INTERFACE I_XTS_Mover_PLC EXTENDS I_CH_Object

{attribute 'OPC.UA.DA.Property' := '1'}
{attribute 'monitoring':='call'}
PROPERTY DefaultAcceleration : LREAL
GET
END_GET
SET
END_SET
END_PROPERTY

{attribute 'OPC.UA.DA.Property' := '1'}
{attribute 'monitoring':='call'}
PROPERTY DefaultDeceleration : LREAL
GET
END_GET
SET
END_SET
END_PROPERTY

{attribute 'OPC.UA.DA.Property' := '1'}
{attribute 'monitoring':='call'}
PROPERTY DefaultJerk : LREAL
GET
END_GET
SET
END_SET
END_PROPERTY

{attribute 'monitoring':='call'}
PROPERTY DrivenDistance : LREAL
GET
END_GET
END_PROPERTY

(*The _ PLC interface provides the user with a simplified interface for commanding between the stations. Sometimes, however, this is not enough. 
Either you get the corresponding interface with the __Queryinterface or you can get full access with this property.*)
PROPERTY FullAccess : I_XTS_Mover
GET
END_GET
END_PROPERTY

{attribute 'monitoring':='call'}
PROPERTY LagDistance : LREAL
GET
END_GET
END_PROPERTY

{attribute 'monitoring':='call'}
PROPERTY LastCmdTargedGap : LREAL
GET
END_GET
END_PROPERTY

{attribute 'monitoring':='call'}
PROPERTY LUID : STRING
GET
END_GET
END_PROPERTY

{attribute 'monitoring':='call'}
PROPERTY PositionOnTrack : LREAL
GET
END_GET
END_PROPERTY

{attribute 'monitoring':='call'}
PROPERTY PUBLIC ProductData : I_XTS_ProductData
GET
END_GET
SET
END_SET
END_PROPERTY

{attribute 'monitoring':='call'}
PROPERTY SetVelocity : LREAL
GET
END_GET
END_PROPERTY

{attribute 'monitoring':='call'}
PROPERTY TargedStation : STRING
GET
END_GET
END_PROPERTY

{attribute 'monitoring':='call'}
PROPERTY UtilityMover : I_TcIoXtsXpuMover
GET
END_GET
END_PROPERTY

END_INTERFACE

(* stored: Version 1.1.0.1, ProductVersion 3.1.4024.12
   Itf I_XTS_Mover_PLC: Id {e47f7de2-f04a-480e-a2ce-8f8f5f0b1a53}
   Property DefaultAcceleration: Id {536791b8-3d03-4e24-a9a7-7540cfae8367}
   Get Get: Id {1442cbe0-f6bc-4f20-91ce-d856c4f7ed62}
   Set Set: Id {ef6db4b8-abe4-4d48-bfb6-b7de2fad2f79}
   Property DefaultDeceleration: Id {9b0d8ce8-a83e-4e2f-a34b-1e46d9561ed8}
   Get Get: Id {8890d087-383c-4b19-9bbf-da61ee0cf101}
   Set Set: Id {4f84c216-f65c-4b2f-b78a-816f68ad9c4a}
   Property DefaultJerk: Id {43968ade-22e7-424f-9fef-d8b8eb4e399e}
   Get Get: Id {7ce9d8a0-38c3-40cc-a375-2892d3f2be8f}
   Set Set: Id {c4d83fa1-caec-47ba-b7ad-4f2729ed75a1}
   Property DrivenDistance: Id {3cdb7f76-6530-45de-884c-f86f69110c1b}
   Get Get: Id {26d92d4a-b4ba-40ce-a7ed-41fcb1369698}
   Property FullAccess: Id {b4794be4-1985-4c4e-aea4-f3bc2f43fe10}
   Get Get: Id {69594b54-a893-46ed-8f3d-c3d54a355990}
   Property LagDistance: Id {b10a5231-09c5-4e83-9ade-98b2be0f8351}
   Get Get: Id {71ef1ad3-0d38-4696-83d1-cf2613b1224d}
   Property LastCmdTargedGap: Id {dbe258f2-3771-42b6-8ba5-29aba506a40b}
   Get Get: Id {18c52b15-646e-4d6f-bf50-b3c739ba8cef}
   Property LUID: Id {207f3dfb-349c-4050-8a27-14772762c31c}
   Get Get: Id {1d565dfc-c9d9-41b4-9a6f-0d83a8a7b355}
   Property PositionOnTrack: Id {e2f77ef3-bbcd-4011-b83c-ce731f495df1}
   Get Get: Id {02b3a8c5-8936-48b3-8f46-8c4dcacfd3ad}
   Property ProductData: Id {e1cb3e8f-1891-4b79-a583-c3f52b72eb8f}
   Get Get: Id {27257a62-8003-4c32-afd4-d3be10359131}
   Set Set: Id {7ca6fde4-535c-479b-a95f-1cd153754543}
   Property SetVelocity: Id {0fcebf09-5353-4bc6-94db-874fad70e86e}
   Get Get: Id {9177b27b-2395-4ac2-a6a7-4a9fbfe3a148}
   Property TargedStation: Id {6ef8f05b-c662-4f85-a1cd-beee94d5369e}
   Get Get: Id {e69626a6-6b37-462f-9cdf-9ac5c6feeafb}
   Property UtilityMover: Id {e026d070-4648-48b6-a50c-d473e07f53a4}
   Get Get: Id {67092823-6484-4ad2-9e91-d73dc2770cbf} *)
